{attribute 'GeneratedUsingTerminal: AX8206-0100-0102-0102'}
{attribute addProperty BoxType "AX8206-0100-0102-0102"}
{attribute addProperty Id "EtcSlaveTerminalBaseDeviceDevice_6E2575772Device_SafetyDevice_Safety_C21945A160Ch_ACh_A_D18C6F1622Ch_BCh_B_647F9A0C22WcStateAT %I*WcState_B516A2644InfoDataAT %I*InfoData_386C00A526"}
{attribute addProperty CRC "4121339909"}
{attribute addProperty Size "136"}
TYPE AX8206_F5A6A805 EXTENDS EtcSlaveTerminalBase :
STRUCT
	{attribute addProperty Name "Device"}
	Device : Device_6E257577;
	{attribute addProperty Name "Device_Safety"}
	Device_Safety : Device_Safety_C21945A1;
	{attribute addProperty Name "Ch_A"}
	Ch_A : Ch_A_D18C6F16;
	{attribute addProperty Name "Ch_B"}
	Ch_B : Ch_B_647F9A0C;
	{attribute addProperty Name "WcState"}
	WcState : WcState_B516A264;
	{attribute addProperty Name "InfoData"}
	InfoData : InfoData_386C00A5;
END_STRUCT
END_TYPE

(* stored: Version 1.2.0.0, ProductVersion 3.1.4024.9
   DUT AX8206_F5A6A805: Id {5ef4ba9c-9c26-4f77-b15e-f8b7fac6c36a} *)
